(* IEC 61131-3 sources: programs/VI-54/VI-54_20171205/VI-54_20171205/Stations/Screen/LseClass170718/Class/EventTitleLine, 1 file *)

(* ---- EventTitleLine.st ---- *)
(*!
<Class
	Name               = "EventTitleLine"
	Revision           = "1.0"
	RealtimeTask       = "false"
	CyclicTask         = "false"
	BackgroundTask     = "false"
	Sigmatek           = "false"
	OSInterface        = "false"
	HighPriority       = "false"
	Automatic          = "false"
	UpdateMode         = "Prescan"
	SharedCommandTable = "true"
	Objectsize         = "(540,240)"
	Comment            = "class for drawing the title line of the EventJournal">
	<Channels>
	</Channels>
	<RevDoku>
		<Owner Author="KaiAnd"/>
		<Dokumentation Revision="1.0" Date="2016-05-11" Author="KaiAnd" Company="Sigmatek" Description="start release"/>
	</RevDoku>
	<Network Name="EventTitleLine">
		<!-- List of Components in this network -->
		<Components>
			<Object
				Name       = "_base"
				Class      = "TitleLine"
				Position   = "(218,120)"
				Visualized = "true"
				Remotely   = "true">
				<Channels>
					<Server Name="Refresh"/>
					<Server Name="Server0"/>
					<Client Name="ColumnChoice"/>
					<Client Name="coSystemLogging"/>
					<Client Name="Lse"/>
				</Channels>
			</Object>
		</Components>
		<Comments>
		</Comments>
		<!-- List of Connections in this network -->
		<Connections>
			<Connection Source="this.Server0" Destination="_base.Server0" Vertices="(942,210),(770,210),"/>
			<Connection Source="this.Refresh" Destination="_base.Refresh" Vertices="(942,270),(770,270),"/>
			<Connection Source="_base.Lse" Destination="this.Lse" Vertices="(218,210),(30,210),(38,210),"/>
			<Connection Source="_base.ColumnChoice" Destination="this.ColumnChoice" Vertices="(218,270),(38,270),"/>
			<Connection Source="_base.coSystemLogging" Destination="this.coSystemLogging" Vertices="(218,330),(38,330),"/>
		</Connections>
		<!-- Headerfiles -->
		<Options>
		</Options>
	</Network>
</Class>
*)
#pragma using TitleLine

EventTitleLine : CLASS
: TitleLine
  //Servers:
  //Clients:
  //Variables:
  //Functions:
				//! <Function Comment="Draws the column texts." Name="DrawHeader"/>
	FUNCTION VIRTUAL DrawHeader
		VAR_INPUT
			pio 	: ^_IO;			//! <Variable Comment="Pointer to the _IO information." Name="DrawHeader.pio"/>
		END_VAR
		VAR_OUTPUT
			bSuccessful 	: BOOL;			//! <Variable Comment="TRUE..Ok&#13;&#10;FALSE..Pointer pio was NIL" Name="DrawHeader.bSuccessful"/>
		END_VAR;
  //Tables:
	FUNCTION @STD
		VAR_OUTPUT
			ret_code	: CONFSTATES;
		END_VAR;
	FUNCTION GLOBAL TAB @CT_;
END_CLASS;

FUNCTION VIRTUAL EventTitleLine::DrawHeader
	VAR_INPUT
		pio 	: ^_IO;
	END_VAR
	VAR_OUTPUT
		bSuccessful 	: BOOL;
	END_VAR

  VAR
    pString     : ^_CHAR;
    tmpRoom     : _ROOM;
    fieldHight  : INT;
    fontWidth   : UINT;
    fontHight   : UINT;
  END_VAR

  // Übergabeparameter prüfen
  if pio = NIL then
    bSuccessful := false;
    return;
  else
    bSuccessful := true;
  end_if;

  // Bestimmen der Position des Texts (Zentriert im Feld)
  fieldHight := pio^.room.xy2.y - pio^.room.xy1.y;
  font_size(x0:=pio^.font, p1:=#fontWidth, p2:=#fontHight);

  tmpRoom.xy1.x := ScrollOffset - 1;
  tmpRoom.xy1.y := pio^.room.xy1.y + ((fieldHight / 2) - (fontHight$INT / 2));
  tmpRoom.xy2.x := ScrollOffset-1;
  tmpRoom.xy2.y := tmpRoom.xy1.y + fontHight$INT;

  // Prüfen ob Text der Spalte1 dargestellt werden soll
  //-----------------------------------------------------------------------------------------
  if ColumnChoice AND 2#000001 then

    // Text aus Textschema holen
    pString$^void := NewDoScheme(x0 := TEXTSCHEME,
                                 x1 := 0,
                                 x2 := ExtVisPara.ParaTextscheme.no);
    if pString = NIL then
      if (IsCon_coSystemLogging = True) then    // KaiAnd
        coSystemLogging.LogEventText("UserListTitel::DrawHeader(): Keinen Text (Eventzeit) gefunden");
      end_if;
    else
      // Koordinaten bestimmen
      tmpRoom.xy1.x := tmpRoom.xy1.x + 5;
      tmpRoom.xy2.x := tmpRoom.xy1.x + to_int(aColumnWidths[0]) - 5;

      // Text ausgeben
      OutTextAlign( p0 := pString,
                    x1 := 0,
                    p1 := #tmpRoom,
                    x2 := pio^.font,
                    x3 := T_SOLID OR T_COPY OR T_PROP OR T_CENTERBOUND OR T_MIDBOUND, // KaiAnd; instead of "pio^.attrib"
                    x9 := _DEFFRAME,
                    x4 := pio^.coltxt,
                    x5 := INVISIBLE,
                    x6 := NIL$_COLOR,
                    x7 := sizeof(_CHAR));
    end_if;

  end_if;

  // Prüfen ob Text der Spalte2 dargestellt werden soll
  //-----------------------------------------------------------------------------------------
  if ColumnChoice AND 2#000010 then

    // Text aus Textschema holen
    pString$^void := NewDoScheme(x0 := TEXTSCHEME,
                                 x1 := 1,
                                 x2 := ExtVisPara.ParaTextscheme.no);
    if pString = NIL then
      if (IsCon_coSystemLogging = True) then    // KaiAnd
        coSystemLogging.LogEventText("TitleLine::DrawHeader(): Keinen Text (Eventzeit) gefunden");
      end_if;
    else
      // Koordinaten bestimmen
      tmpRoom.xy1.x := tmpRoom.xy2.x + 5;
      tmpRoom.xy2.x := tmpRoom.xy1.x + to_int(aColumnWidths[1]) - 5;

      // Text ausgeben
      OutTextAlign( p0 := pString,
                    x1 := 0,
                    p1 := #tmpRoom,
                    x2 := pio^.font,
                    x3 := T_SOLID OR T_COPY OR T_PROP OR T_CENTERBOUND OR T_MIDBOUND, // KaiAnd; instead of "pio^.attrib"
                    x9 := _DEFFRAME,
                    x4 := pio^.coltxt,
                    x5 := INVISIBLE,
                    x6 := NIL$_COLOR,
                    x7 := sizeof(_CHAR));
    end_if;

  end_if;

  // Prüfen ob Text der Spalte3 dargestellt werden soll
  //-----------------------------------------------------------------------------------------
  if ColumnChoice AND 2#000100 then

    //Text aus Textschema holen
    pString$^void := NewDoScheme(x0 := TEXTSCHEME,
                                 x1 := 2,
                                 x2 := ExtVisPara.ParaTextscheme.no);
    if pString = NIL then
      if (IsCon_coSystemLogging = True) then    // KaiAnd
        coSystemLogging.LogEventText("TitleLine::DrawHeader(): Keinen Text (Alarmnummer) gefunden");
      end_if;
    else
      // Koordinaten bestimmen
      tmpRoom.xy1.x := tmpRoom.xy2.x + 5;
      tmpRoom.xy2.x := tmpRoom.xy1.x + to_int(aColumnWidths[2]) - 5;

      // Text ausgeben
      OutTextAlign( p0 := pString,
                    x1 := 0,
                    p1 := #tmpRoom,
                    x2 := pio^.font,
                    x3 := T_SOLID OR T_COPY OR T_PROP OR T_CENTERBOUND OR T_MIDBOUND, // KaiAnd; instead of "pio^.attrib"
                    x9 := _DEFFRAME,
                    x4 := pio^.coltxt,
                    x5 := INVISIBLE,
                    x6 := NIL$_COLOR,
                    x7 := sizeof(_CHAR));

    end_if;

  end_if;

  // Prüfen ob Text der Spalte4 dargestellt werden soll
  //-----------------------------------------------------------------------------------------
  if ColumnChoice AND 2#001000 then

    // Text aus Textschema holen
    pString$^void := NewDoScheme(x0 := TEXTSCHEME,
                                 x1 := 3,
                                 x2 := ExtVisPara.ParaTextscheme.no);
    if pString = NIL then
      if (IsCon_coSystemLogging = True) then    // KaiAnd
        coSystemLogging.LogEventText("TitleLine::DrawHeader(): Keinen Text (Accesslevel) gefunden");
      end_if;
    else
      // Koordinaten bestimmen
      tmpRoom.xy1.x := tmpRoom.xy2.x + 5;
      tmpRoom.xy2.x := tmpRoom.xy1.x + to_int(aColumnWidths[3]) - 5;

      // Text ausgeben
      OutTextAlign( p0 := pString,
                    x1 := 0,
                    p1 := #tmpRoom,
                    x2 := pio^.font,
                    x3 := T_SOLID OR T_COPY OR T_PROP OR T_CENTERBOUND OR T_MIDBOUND, // KaiAnd; instead of "pio^.attrib"
                    x9 := _DEFFRAME,
                    x4 := pio^.coltxt,
                    x5 := INVISIBLE,
                    x6 := NIL$_COLOR,
                    x7 := sizeof(_CHAR));
    end_if;

  end_if;

  // Prüfen ob Text der Spalte5 dargestellt werden soll
  //-----------------------------------------------------------------------------------------
  if ColumnChoice AND 2#010000 then

    // Text aus Textschema holen
    pString$^void := NewDoScheme(x0 := TEXTSCHEME,
                                 x1 := 4,
                                 x2 := ExtVisPara.ParaTextscheme.no);
    if pString = NIL then
      if (IsCon_coSystemLogging = True) then    // KaiAnd
        coSystemLogging.LogEventText("TitleLine::DrawHeader(): Keinen Text (Beschreibung) gefunden");
      end_if;
    else
      // Koordinaten bestimmen
      tmpRoom.xy1.x := tmpRoom.xy2.x + 5;
      tmpRoom.xy2.x := tmpRoom.xy1.x + to_int(aColumnWidths[4]) - 5;

      // Text ausgeben
      OutTextAlign( p0 := pString,
                    x1 := 0,
                    p1 := #tmpRoom,
                    x2 := pio^.font,
                    x3 := pio^.attrib,
                    x9 := _DEFFRAME,
                    x4 := pio^.coltxt,
                    x5 := INVISIBLE,
                    x6 := NIL$_COLOR,
                    x7 := sizeof(_CHAR));
    end_if;

  end_if;

  // Prüfen ob Text der Spalte6 dargestellt werden soll
  //-----------------------------------------------------------------------------------------
  if ColumnChoice AND 2#100000 then

    // Text aus Textschema holen
    pString$^void := NewDoScheme(x0 := TEXTSCHEME,
                                 x1 := 5,
                                 x2 := ExtVisPara.ParaTextscheme.no);
    if pString = NIL then
      if (IsCon_coSystemLogging = True) then    // KaiAnd
        coSystemLogging.LogEventText("TitleLine::DrawHeader(): Keinen Text (Beschreibung) gefunden");
      end_if;
    else
      // Koordinaten bestimmen
      tmpRoom.xy1.x := tmpRoom.xy2.x + 5;
      tmpRoom.xy2.x := tmpRoom.xy1.x + to_int(aColumnWidths[5]) - 5;

      // Text ausgeben
      OutTextAlign( p0 := pString,
                    x1 := 0,
                    p1 := #tmpRoom,
                    x2 := pio^.font,
                    x3 := T_LEFTBOUND or T_SOLID or T_PROP or T_COPY or T_MIDBOUND,
                    x9 := _DEFFRAME,
                    x4 := pio^.coltxt,
                    x5 := INVISIBLE,
                    x6 := NIL$_COLOR,
                    x7 := sizeof(_CHAR));
    end_if;

  end_if;

END_FUNCTION
